(* Logix 5000 project; controller cal1615 1756-L62 rev 20.19; software revision 20.05; part 28 of 82 *)
(* tags used below, declared in another part *)
   FAULT : BOOL;   // Fault AFI
   p01_param_fan_zero_speed : REAL;
   p01_param_open_oven_recirc_sp : REAL;
   p01_param_temp_limit : REAL;   // Machine Parameter Maximum Temperature for Fan Operation
   p01_recipe_active : recipe;   // Active Recipe
   p01r02 : routine;   // System Misc Control
   p01r09_open_oven : BOOL;
   p01r09_pb_global_reset : BOOL;   // System Modes PB: Global Fault Reset
   p02_dint_from_hmi : hmi_dint;
   p11r02_shutdown_temp : BOOL;   // Zone 1 Misc Control Safe Shutdown Temperature
   p11r30 : routine;   // Zone 1 Temperature Control
   p12_ai_recirc_rpm : REAL;   // Zone 2 Analog Input Recirc Fan RPM
   p12_ao_recirc_selected_speed : REAL;   // Zone 2 Analog Output Recirc Fan VFD Selected Speed
   p12_di_recirc : acs800_di_normal;   // Zone 2 Digital Inputs Recirc Fan
   p12_di_recirc_fan_mtr_ts : BOOL;   // Zone 2 Digital Input Recirc Fan Motor Thermostat OK
   p12_di_recirc_flow_ok : BOOL;   // Zone 2 Digital Input Recirc Flow OK
   p12_do_recirc : acs800_do_normal;   // Zone 2 Digital Outputs Supply Fan
   p12r01 : routine;   // Zone 2 Main
   p12r02_shutdown_temp : BOOL;   // Zone 2 Misc Control Safe Shutdown Temperature
   p12r20_state : DINT;   // Zone 2 Temperature Control State
   p12r30 : routine;   // Zone 2 Temperature Control
   p12r32 : routine;   // Zone 2 Recirc VFD
   p12r32_fan_pb_stopped : BOOL;   // Zone 2 Recirc VFD Fan Stopped Manually - Prevent Auto Start during Cooldown
   p12r32_pb_start : BOOL;   // Zone 2 Recirc VFD PB: Start
   p12r32_pb_stop : BOOL;   // Zone 2 Recirc VFD PB: Stop
   p12r32_request_auto_run : BOOL;   // Zone 2 Recirc Fan Run Request
   p12r32_run_permissive : BOOL;   // Zone 2 Recirc VFD Run Permissive
   p12r32_timer_fault : TIMER[5];   // Zone 2 Recirc VFD Fault Timer
   p12r32_timer_warning : TIMER[5];   // Zone 2 Supply VFD Warning Timer
   p12r32_vfd_stopped : BOOL;   // Zone 2 Recirc VFD VFD Stopped
   p13_ai_tc01 : REAL;   // Zone 3 Analog Input Control Thermocouple 1
   p13_ai_tc02 : REAL;   // Zone 3 Analog Input Control Thermocouple 2
   p13_dint_to_hmi : DINT[16];   // Zone 3 Temperature Control VFDs On
   p13_param_shutdown_temp : REAL;   // Zone 3 Parameter Zone Shutdown Temperature
   p13r01 : routine;   // Zone 3 Main
   p13r02 : routine;   // Zone 3 Misc Control
   p13r02_fault_exists : BOOL;
   p13r02_not_safe_temp : BOOL;   // Zone 3 Misc Control Zone above Safe Temp
   p13r02_safe_temp : BOOL;   // Zone 3 Misc Control Zone Temperature at Safe Temp
   p13r02_shutdown_temp : BOOL;   // Zone 3 Misc Control Safe Shutdown Temperature
   p13r02_timer_fault : TIMER[4];   // Zone 3 Misc Control Fault Delay
   p13r02_timer_safe_temp : TIMER[2];   // Zone 3 Misc Control Chamber SafeTemperature Dwell
   p13r02_timer_warning : TIMER[4];   // Zone 3 Misc Control Warning Delay
   p13r02_unack_fault : BOOL;   // Zone 3 Misc Control Unacknowledged Fault Exists
   p13r02_unack_warning : BOOL;   // Zone 3 Misc Control Unacknowledged Warning Exists
   p13r02_warning_exists : BOOL;
   p13r03 : routine;   // Zone 3 Input
   p13r04 : routine;   // Zone 3 Output
   p13r05 : routine;   // Zone 3 Dint to HMI
   p13r06 : routine;   // Zone 3 Real to HMI
   p13r07 : routine;   // Zone 3 Alarms
   p13r08 : routine;   // Zone 3 Warnings
   p13r09 : routine;   // Zone 3 Modes
   p13r10 : routine;   // Zone 3
   p13r20 : routine;   // Zone 3 Temp Sequence
   p13r30 : routine;   // Zone 3 Temperature Control
   p13r31 : routine;   // Zone 3 Exhaust VFD
   p13r32 : routine;   // Zone 3 Recirc VFD
   p23r02 : routine;   // Impreg Misc Control
(* P12_Zone_2, continued *)

ROUTINE R32_Recirc_VFD   (* ladder *)
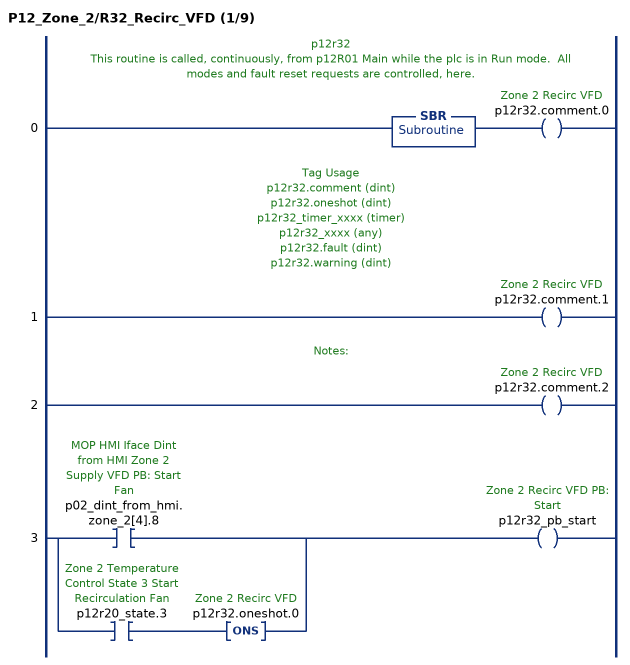
   // p12r32
   // This routine is called, continuously, from p12R01 Main while the plc is in Run mode.  All modes and fault reset requests are controlled, here.
   0: SBR()OTE(p12r32.comment.0);
   // Tag Usage
   // p12r32.comment (dint)
   // p12r32.oneshot (dint)
   // p12r32_timer_xxxx (timer)
   // p12r32_xxxx (any)
   // p12r32.fault (dint)
   // p12r32.warning (dint)
   1: OTE(p12r32.comment.1);
   // Notes:
   2: OTE(p12r32.comment.2);
   3: [XIC(p02_dint_from_hmi.zone_2[4].8) ,XIC(p12r20_state.3) ONS(p12r32.oneshot.0) ]OTE(p12r32_pb_start);
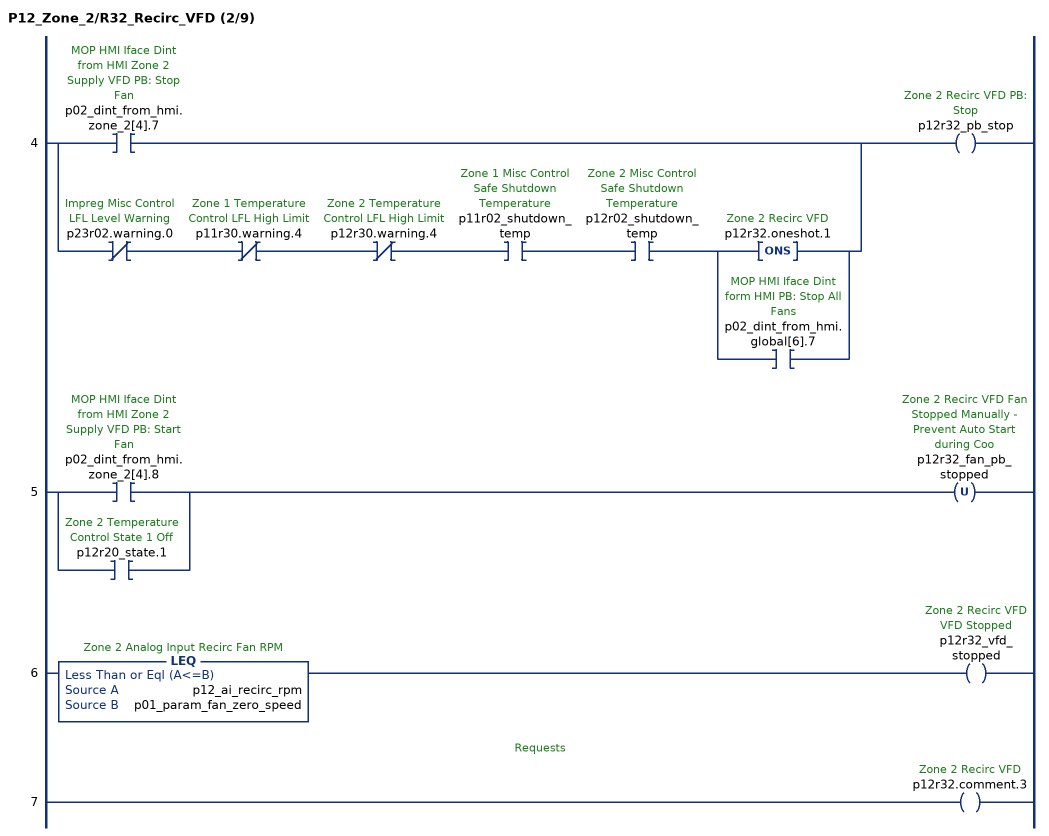
   4: [XIC(p02_dint_from_hmi.zone_2[4].7) ,XIO(p23r02.warning.0) XIO(p11r30.warning.4) XIO(p12r30.warning.4) XIC(p11r02_shutdown_temp) XIC(p12r02_shutdown_temp) [ONS(p12r32.oneshot.1) ,XIC(p02_dint_from_hmi.global[6].7) ] ]OTE(p12r32_pb_stop);
   5: [XIC(p02_dint_from_hmi.zone_2[4].8) ,XIC(p12r20_state.1) ]OTU(p12r32_fan_pb_stopped);
   6: LEQ(p12_ai_recirc_rpm,p01_param_fan_zero_speed)OTE(p12r32_vfd_stopped);
   // Requests
   7: OTE(p12r32.comment.3);
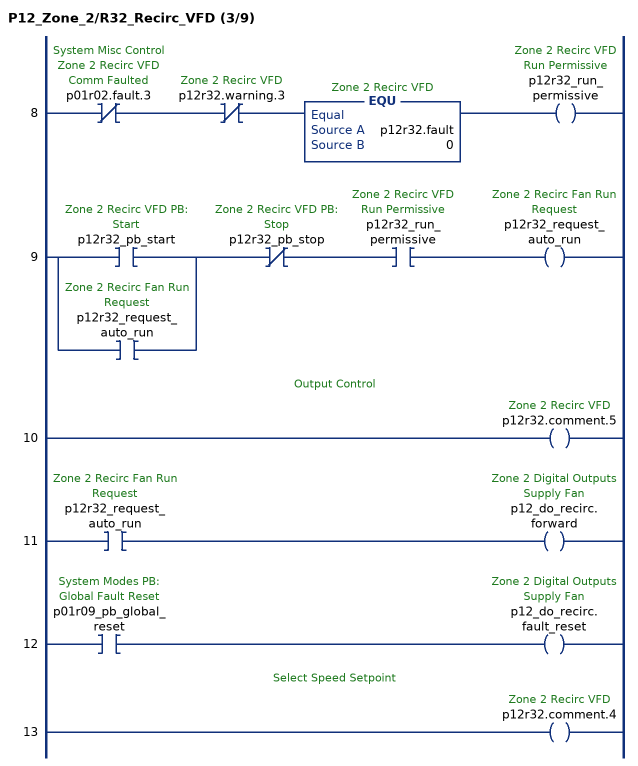
   8: XIO(p01r02.fault.3)XIO(p12r32.warning.3)EQU(p12r32.fault,0)OTE(p12r32_run_permissive);
   9: [XIC(p12r32_pb_start) ,XIC(p12r32_request_auto_run) ]XIO(p12r32_pb_stop)XIC(p12r32_run_permissive)OTE(p12r32_request_auto_run);
   // Output Control
   10: OTE(p12r32.comment.5);
   11: XIC(p12r32_request_auto_run)OTE(p12_do_recirc.forward);
   12: XIC(p01r09_pb_global_reset)OTE(p12_do_recirc.fault_reset);
   // Select Speed Setpoint
   13: OTE(p12r32.comment.4);
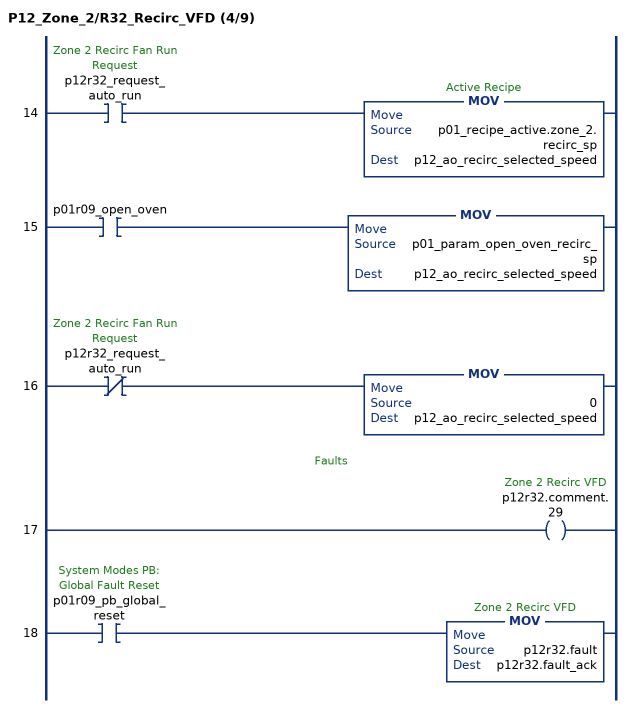
   14: XIC(p12r32_request_auto_run)MOV(p01_recipe_active.zone_2.recirc_sp,p12_ao_recirc_selected_speed);
   15: XIC(p01r09_open_oven)MOV(p01_param_open_oven_recirc_sp,p12_ao_recirc_selected_speed);
   16: XIO(p12r32_request_auto_run)MOV(0,p12_ao_recirc_selected_speed);
   // Faults
   17: OTE(p12r32.comment.29);
   18: XIC(p01r09_pb_global_reset)MOV(p12r32.fault,p12r32.fault_ack);
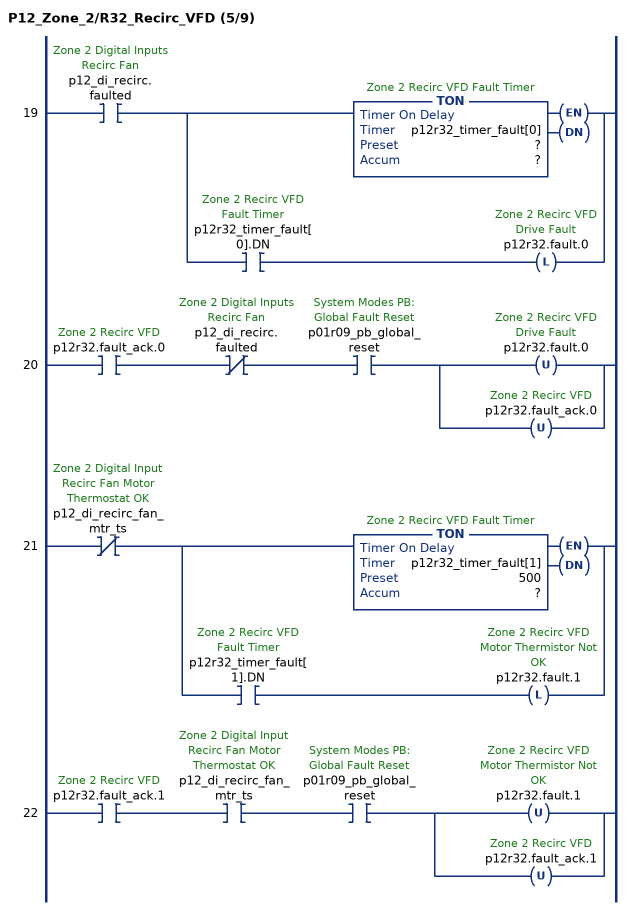
   19: XIC(p12_di_recirc.faulted)[TON(p12r32_timer_fault[0],?,?) ,XIC(p12r32_timer_fault[0].DN) OTL(p12r32.fault.0) ];
   20: XIC(p12r32.fault_ack.0)XIO(p12_di_recirc.faulted)XIC(p01r09_pb_global_reset)[OTU(p12r32.fault.0) ,OTU(p12r32.fault_ack.0) ];
   21: XIO(p12_di_recirc_fan_mtr_ts)[TON(p12r32_timer_fault[1],?,?) ,XIC(p12r32_timer_fault[1].DN) OTL(p12r32.fault.1) ];
   22: XIC(p12r32.fault_ack.1)XIC(p12_di_recirc_fan_mtr_ts)XIC(p01r09_pb_global_reset)[OTU(p12r32.fault.1) ,OTU(p12r32.fault_ack.1) ];
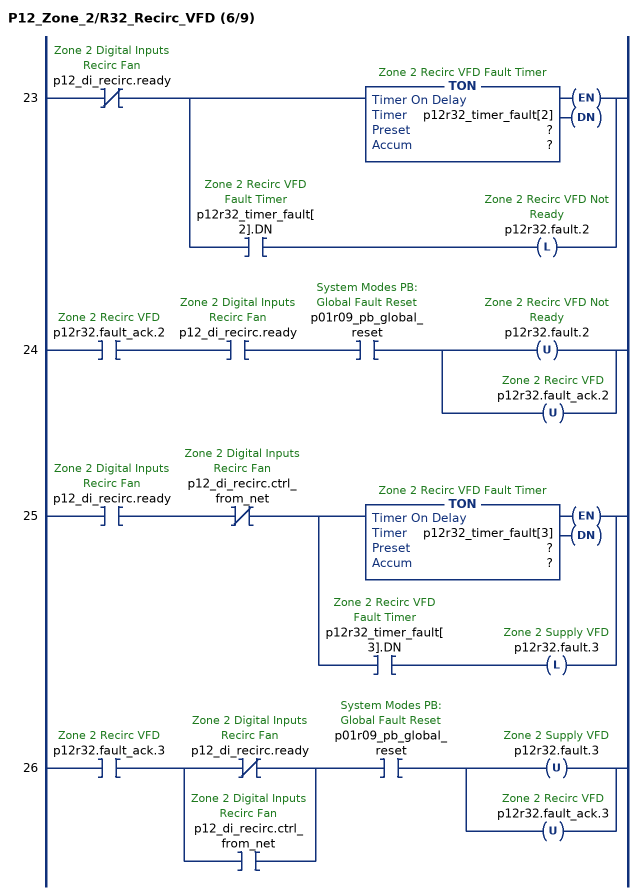
   23: XIO(p12_di_recirc.ready)[TON(p12r32_timer_fault[2],?,?) ,XIC(p12r32_timer_fault[2].DN) OTL(p12r32.fault.2) ];
   24: XIC(p12r32.fault_ack.2)XIC(p12_di_recirc.ready)XIC(p01r09_pb_global_reset)[OTU(p12r32.fault.2) ,OTU(p12r32.fault_ack.2) ];
   25: XIC(p12_di_recirc.ready)XIO(p12_di_recirc.ctrl_from_net)[TON(p12r32_timer_fault[3],?,?) ,XIC(p12r32_timer_fault[3].DN) OTL(p12r32.fault.3) ];
   26: XIC(p12r32.fault_ack.3)[XIO(p12_di_recirc.ready) ,XIC(p12_di_recirc.ctrl_from_net) ]XIC(p01r09_pb_global_reset)[OTU(p12r32.fault.3) ,OTU(p12r32.fault_ack.3) ];
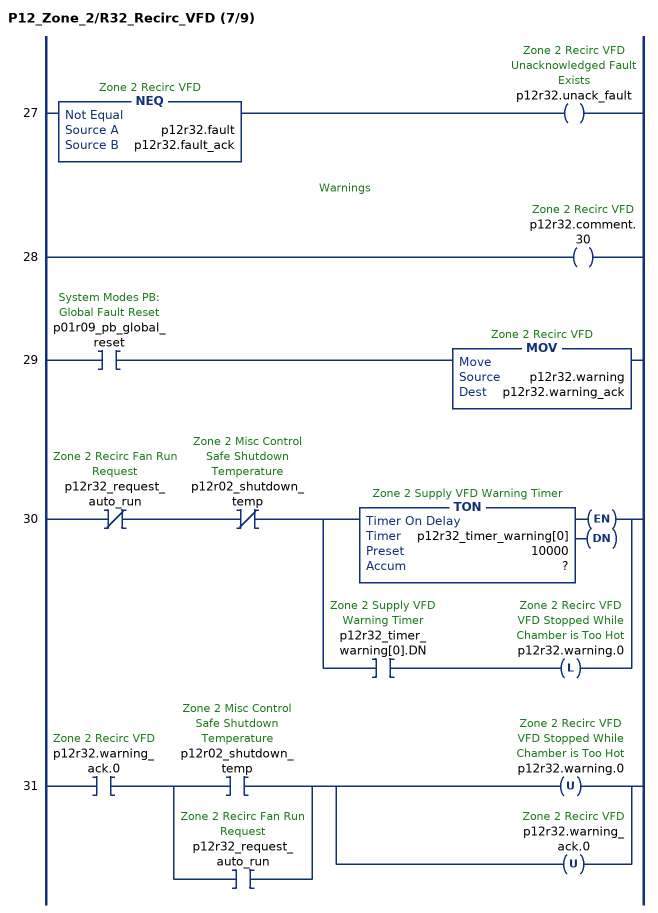
   27: NEQ(p12r32.fault,p12r32.fault_ack)OTE(p12r32.unack_fault);
   // Warnings
   28: OTE(p12r32.comment.30);
   29: XIC(p01r09_pb_global_reset)MOV(p12r32.warning,p12r32.warning_ack);
   30: XIO(p12r32_request_auto_run)XIO(p12r02_shutdown_temp)[TON(p12r32_timer_warning[0],?,?) ,XIC(p12r32_timer_warning[0].DN) OTL(p12r32.warning.0) ];
   31: XIC(p12r32.warning_ack.0)[XIC(p12r02_shutdown_temp) ,XIC(p12r32_request_auto_run) ][OTU(p12r32.warning.0) ,OTU(p12r32.warning_ack.0) ];
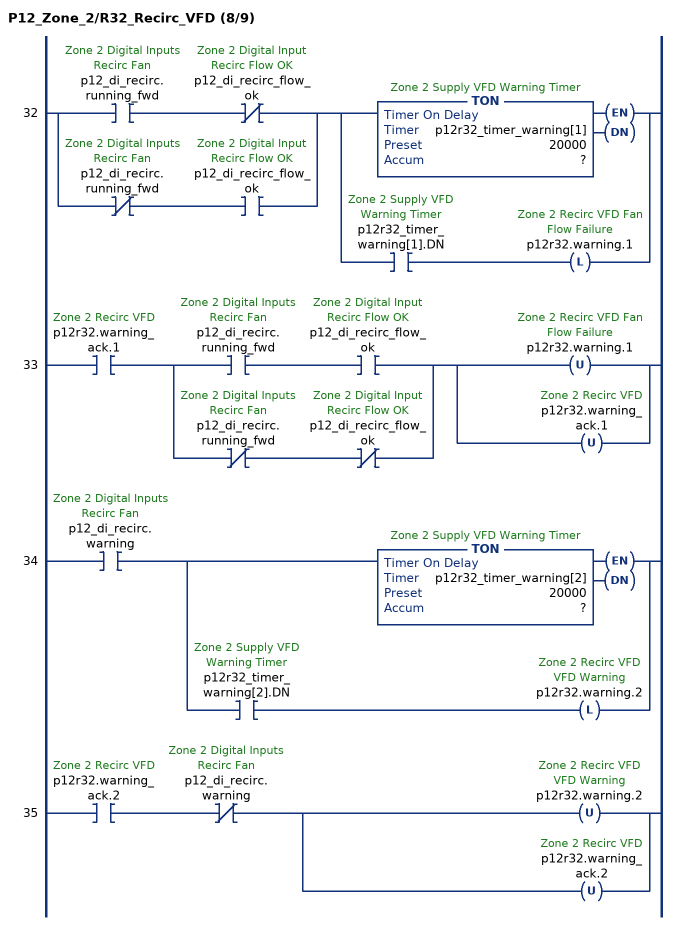
   32: [XIC(p12_di_recirc.running_fwd) XIO(p12_di_recirc_flow_ok) ,XIO(p12_di_recirc.running_fwd) XIC(p12_di_recirc_flow_ok) ][TON(p12r32_timer_warning[1],?,?) ,XIC(p12r32_timer_warning[1].DN) OTL(p12r32.warning.1) ];
   33: XIC(p12r32.warning_ack.1)[XIC(p12_di_recirc.running_fwd) XIC(p12_di_recirc_flow_ok) ,XIO(p12_di_recirc.running_fwd) XIO(p12_di_recirc_flow_ok) ][OTU(p12r32.warning.1) ,OTU(p12r32.warning_ack.1) ];
   34: XIC(p12_di_recirc.warning)[TON(p12r32_timer_warning[2],?,?) ,XIC(p12r32_timer_warning[2].DN) OTL(p12r32.warning.2) ];
   35: XIC(p12r32.warning_ack.2)XIO(p12_di_recirc.warning)[OTU(p12r32.warning.2) ,OTU(p12r32.warning_ack.2) ];
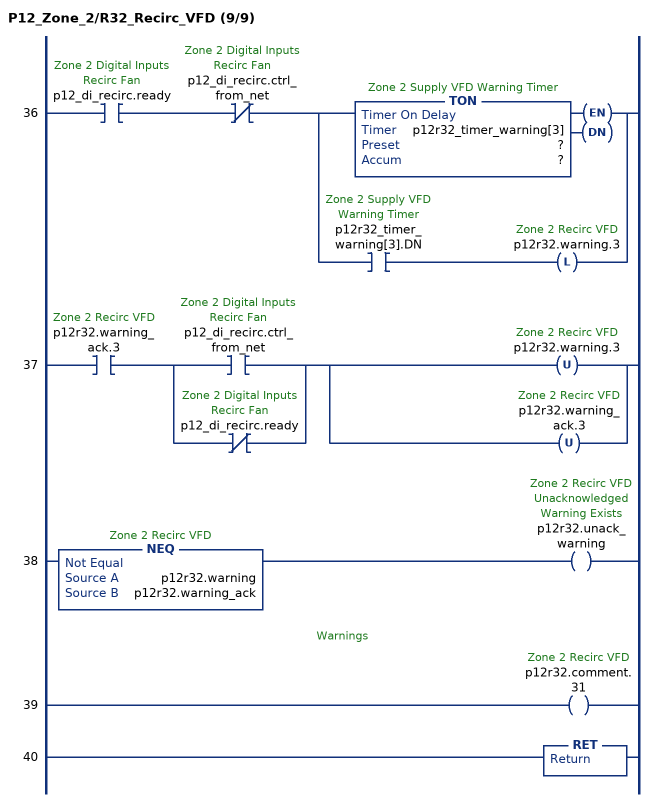
   36: XIC(p12_di_recirc.ready)XIO(p12_di_recirc.ctrl_from_net)[TON(p12r32_timer_warning[3],?,?) ,XIC(p12r32_timer_warning[3].DN) OTL(p12r32.warning.3) ];
   37: XIC(p12r32.warning_ack.3)[XIC(p12_di_recirc.ctrl_from_net) ,XIO(p12_di_recirc.ready) ][OTU(p12r32.warning.3) ,OTU(p12r32.warning_ack.3) ];
   38: NEQ(p12r32.warning,p12r32.warning_ack)OTE(p12r32.unack_warning);
   // Warnings
   39: OTE(p12r32.comment.31);
   40: RET();
END_ROUTINE
END_PROGRAM

PROGRAM P13_Zone_3   (* main routine R01_Main *)

ROUTINE R01_Main   (* ladder *)
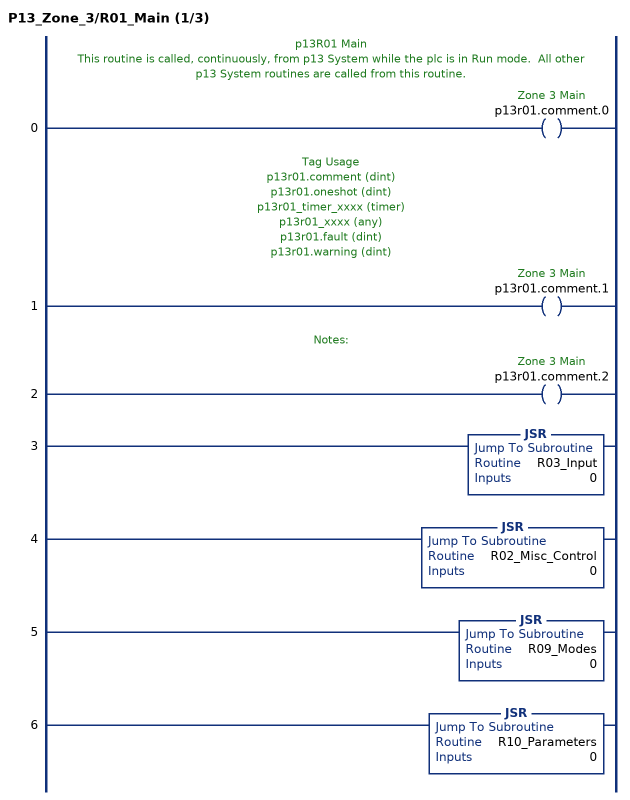
   // p13R01 Main
   // This routine is called, continuously, from p13 System while the plc is in Run mode.  All other p13 System routines are called from this routine.
   0: OTE(p13r01.comment.0);
   // Tag Usage
   // p13r01.comment (dint)
   // p13r01.oneshot (dint)
   // p13r01_timer_xxxx (timer)
   // p13r01_xxxx (any)
   // p13r01.fault (dint)
   // p13r01.warning (dint)
   1: OTE(p13r01.comment.1);
   // Notes:
   2: OTE(p13r01.comment.2);
   3: JSR(R03_Input,0);
   4: JSR(R02_Misc_Control,0);
   5: JSR(R09_Modes,0);
   6: JSR(R10_Parameters,0);
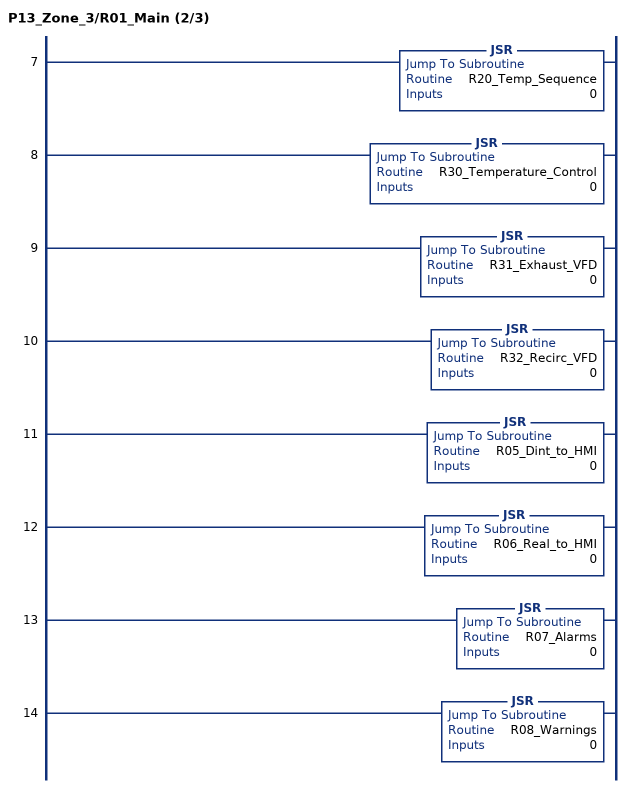
   7: JSR(R20_Temp_Sequence,0);
   8: JSR(R30_Temperature_Control,0);
   9: JSR(R31_Exhaust_VFD,0);
   10: JSR(R32_Recirc_VFD,0);
   11: JSR(R05_Dint_to_HMI,0);
   12: JSR(R06_Real_to_HMI,0);
   13: JSR(R07_Alarms,0);
   14: JSR(R08_Warnings,0);
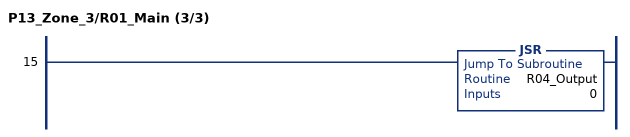
   15: JSR(R04_Output,0);
END_ROUTINE

ROUTINE R02_Misc_Control   (* ladder *)
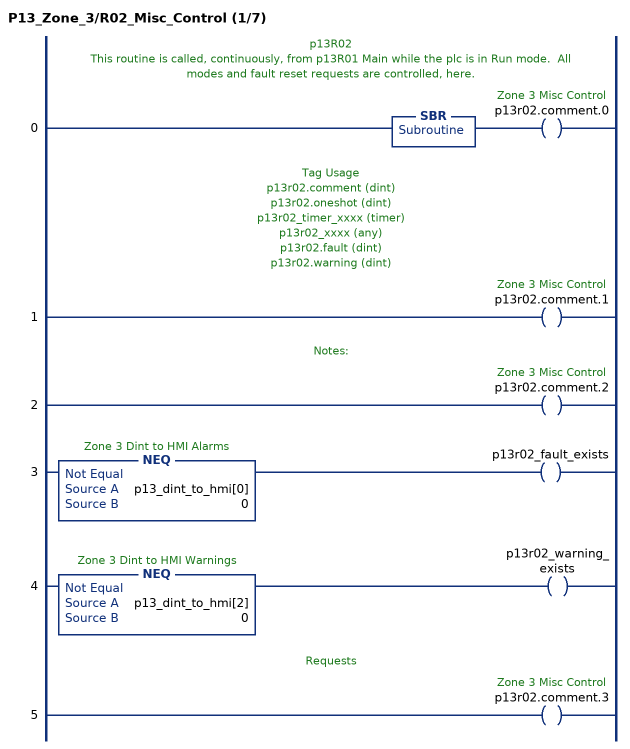
   // p13R02
   // This routine is called, continuously, from p13R01 Main while the plc is in Run mode.  All modes and fault reset requests are controlled, here.
   0: SBR()OTE(p13r02.comment.0);
   // Tag Usage
   // p13r02.comment (dint)
   // p13r02.oneshot (dint)
   // p13r02_timer_xxxx (timer)
   // p13r02_xxxx (any)
   // p13r02.fault (dint)
   // p13r02.warning (dint)
   1: OTE(p13r02.comment.1);
   // Notes:
   2: OTE(p13r02.comment.2);
   3: NEQ(p13_dint_to_hmi[0],0)OTE(p13r02_fault_exists);
   4: NEQ(p13_dint_to_hmi[2],0)OTE(p13r02_warning_exists);
   // Requests
   5: OTE(p13r02.comment.3);
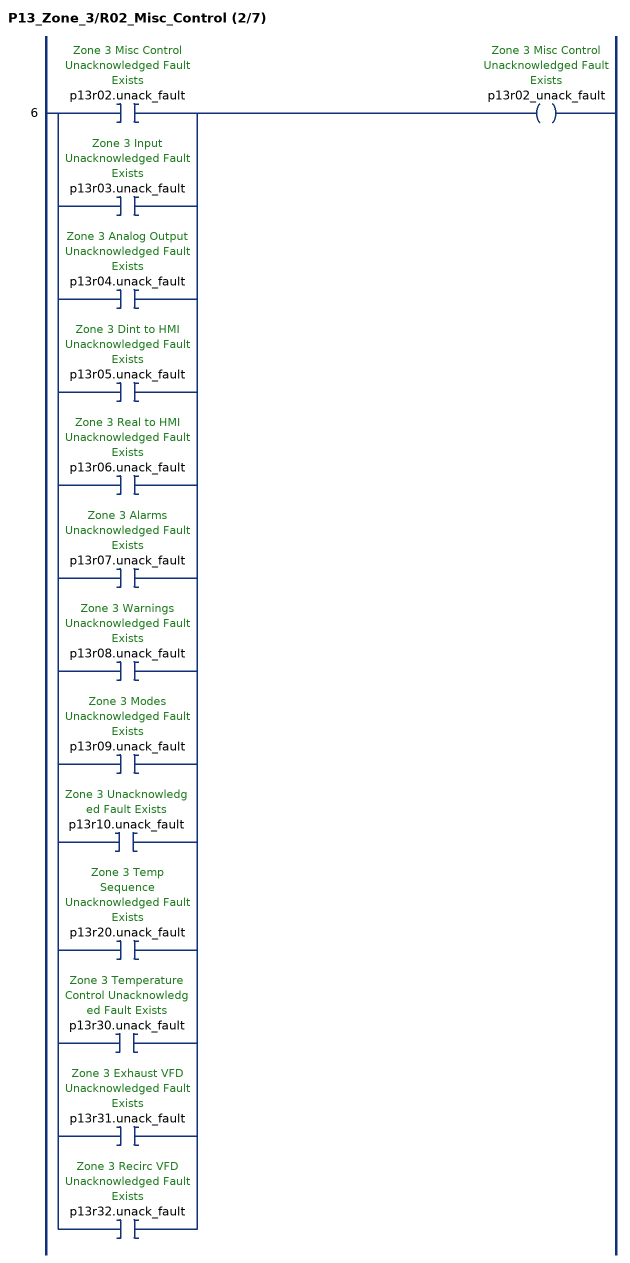
   6: [XIC(p13r02.unack_fault) ,XIC(p13r03.unack_fault) ,XIC(p13r04.unack_fault) ,XIC(p13r05.unack_fault) ,XIC(p13r06.unack_fault) ,XIC(p13r07.unack_fault) ,XIC(p13r08.unack_fault) ,XIC(p13r09.unack_fault) ,XIC(p13r10.unack_fault) ,XIC(p13r20.unack_fault) ,XIC(p13r30.unack_fault) ,XIC(p13r31.unack_fault) ,XIC(p13r32.unack_fault) ]OTE(p13r02_unack_fault);
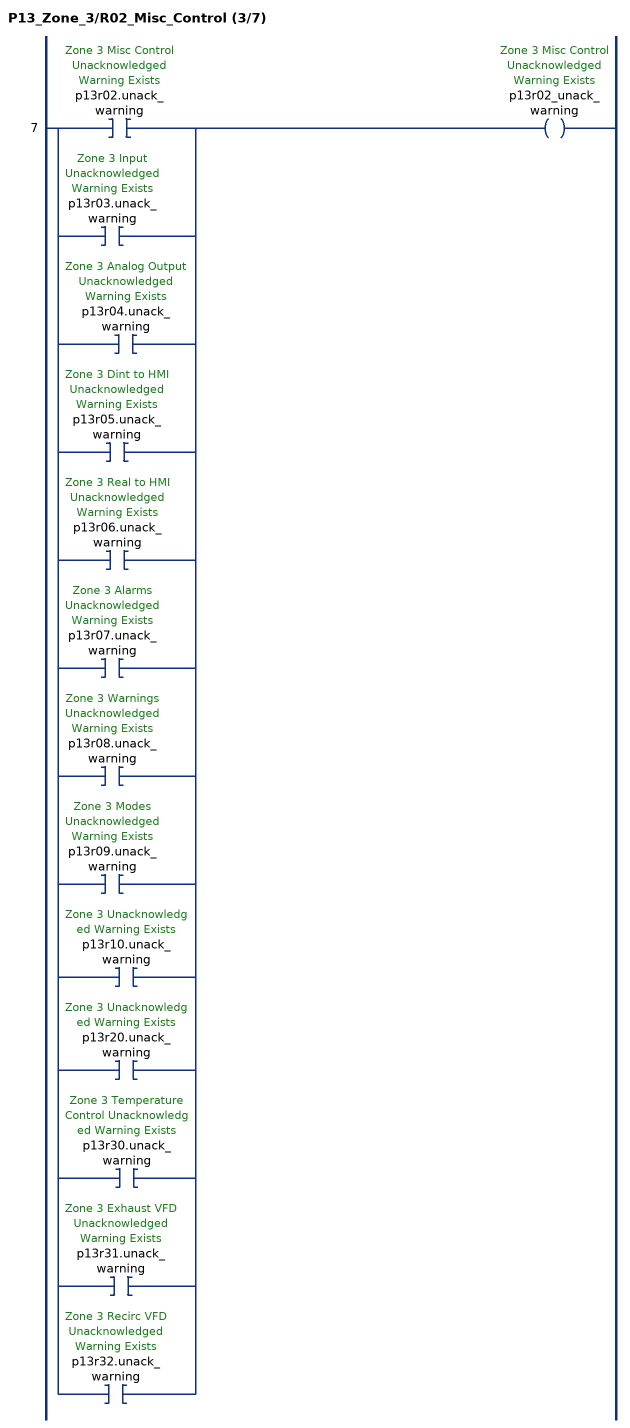
   7: [XIC(p13r02.unack_warning) ,XIC(p13r03.unack_warning) ,XIC(p13r04.unack_warning) ,XIC(p13r05.unack_warning) ,XIC(p13r06.unack_warning) ,XIC(p13r07.unack_warning) ,XIC(p13r08.unack_warning) ,XIC(p13r09.unack_warning) ,XIC(p13r10.unack_warning) ,XIC(p13r20.unack_warning) ,XIC(p13r30.unack_warning) ,XIC(p13r31.unack_warning) ,XIC(p13r32.unack_warning) ]OTE(p13r02_unack_warning);
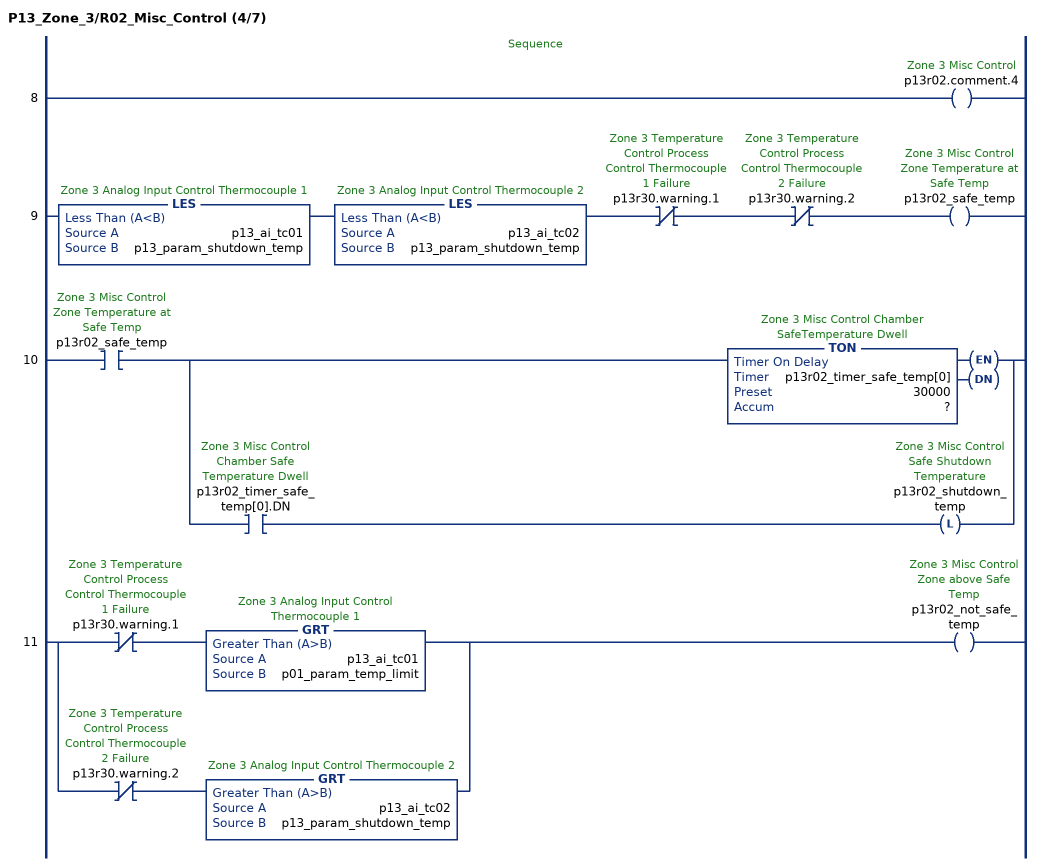
   // Sequence
   8: OTE(p13r02.comment.4);
   9: LES(p13_ai_tc01,p13_param_shutdown_temp)LES(p13_ai_tc02,p13_param_shutdown_temp)XIO(p13r30.warning.1)XIO(p13r30.warning.2)OTE(p13r02_safe_temp);
   10: XIC(p13r02_safe_temp)[TON(p13r02_timer_safe_temp[0],?,?) ,XIC(p13r02_timer_safe_temp[0].DN) OTL(p13r02_shutdown_temp) ];
   11: [XIO(p13r30.warning.1) GRT(p13_ai_tc01,p01_param_temp_limit) ,XIO(p13r30.warning.2) GRT(p13_ai_tc02,p13_param_shutdown_temp) ]OTE(p13r02_not_safe_temp);
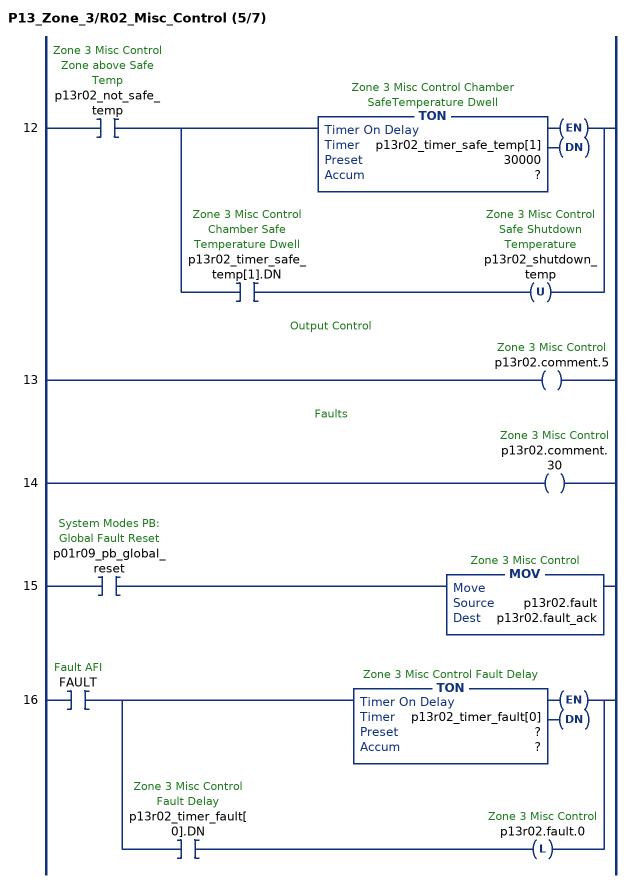
   12: XIC(p13r02_not_safe_temp)[TON(p13r02_timer_safe_temp[1],?,?) ,XIC(p13r02_timer_safe_temp[1].DN) OTU(p13r02_shutdown_temp) ];
   // Output Control
   13: OTE(p13r02.comment.5);
   // Faults
   14: OTE(p13r02.comment.30);
   15: XIC(p01r09_pb_global_reset)MOV(p13r02.fault,p13r02.fault_ack);
   16: XIC(FAULT)[TON(p13r02_timer_fault[0],?,?) ,XIC(p13r02_timer_fault[0].DN) OTL(p13r02.fault.0) ];
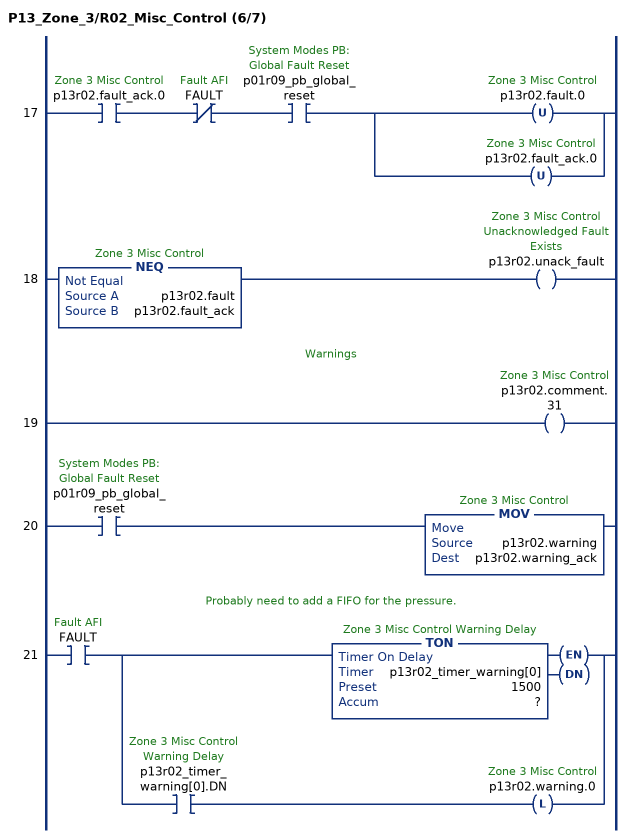
   17: XIC(p13r02.fault_ack.0)XIO(FAULT)XIC(p01r09_pb_global_reset)[OTU(p13r02.fault.0) ,OTU(p13r02.fault_ack.0) ];
   18: NEQ(p13r02.fault,p13r02.fault_ack)OTE(p13r02.unack_fault);
   // Warnings
   19: OTE(p13r02.comment.31);
   20: XIC(p01r09_pb_global_reset)MOV(p13r02.warning,p13r02.warning_ack);
   // Probably need to add a FIFO for the pressure.
   21: XIC(FAULT)[TON(p13r02_timer_warning[0],?,?) ,XIC(p13r02_timer_warning[0].DN) OTL(p13r02.warning.0) ];
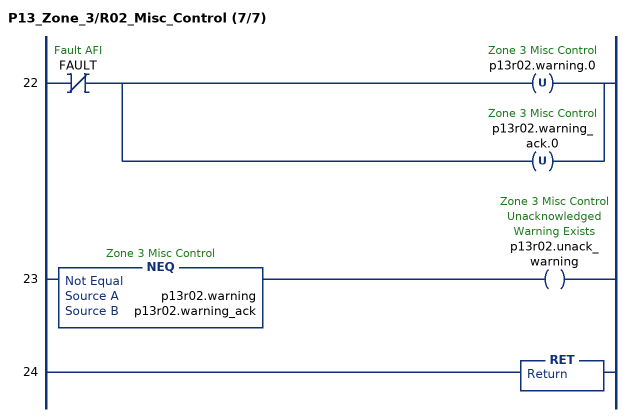
   22: XIO(FAULT)[OTU(p13r02.warning.0) ,OTU(p13r02.warning_ack.0) ];
   23: NEQ(p13r02.warning,p13r02.warning_ack)OTE(p13r02.unack_warning);
   24: RET();
END_ROUTINE
